// TIA Portal V17 export
// export: Created 2023-12-09T21:22:34.4030221Z, ExportSetting WithDefaults, DisplayName Totally Integrated Automation Portal, DisplayVersion V17, DisplayName TIA Portal Openness, DisplayVersion V17, DisplayName TIA Portal Teamcenter Gateway, DisplayVersion V17, DisplayName TIA Portal Version Control Interface, DisplayVersion V17, DisplayName STEP 7 Professional, DisplayVersion V17, DisplayName STEP 7 Safety, DisplayVersion V17, DisplayName WinCC Advanced / Unified PC, DisplayVersion V17
DATA_BLOCK "TRCV_C_DB_1"   // DB6
// stored: AutoNumber true, InstanceOfName TRCV_C, OfSystemLibElement TRCV_C, OfSystemLibVersion 2.1
"TRCV_C"
   // VAR_INPUT
   //    EN_R : Bool;
   //    CONT : Bool;
   //    LEN : UInt;
   // END_VAR
   // VAR_OUTPUT
   //    DONE : Bool;
   //    BUSY : Bool;
   //    ERROR : Bool;
   //    STATUS : Word;
   //    RCVD_LEN : UInt;
   // END_VAR
   // VAR_IN_OUT
   //    CONNECT : TCON_Param;
   //    DATA : Variant;
   //    COM_RST : Bool;
   // END_VAR
   // VAR
   //    sb_FIRSTSTART : Bool;
   //    sb_COMRST : Bool;
   //    sb_CON_EST : Bool;
   //    sb_STARTFB : Bool;
   //    sw_ConID : CONN_OUC;
   //    si_STATE : UInt;
   //    si_JOB : UInt;
   //    s_TCON { S7_SetPoint := 'True'} : TCON;
   //    s_TRCV { S7_SetPoint := 'True'} : TRCV;
   //    s_TDISCON { S7_SetPoint := 'True'} : TDISCON;
   // END_VAR
BEGIN
END_DATA_BLOCK
